(* Logix 5000 project; controller KTC_lab3 vendor 1 type 14 code 149 rev 30.11; software revision 30.00 *)

TASK MainTask (continuous, watchdog 500 ms) : MainProgram

MODULES
   Local : vendor 1 type 14 code 149 (Compact 0, rev 30.11)
      Discrete_IO : Embedded (Compact 1, rev 3.1, Output RPI 20 ms)
END_MODULES

PROGRAM MainProgram   (* main routine MainRoutine *)
VAR
   B3_1 : BOOL;   // SHUT DOWN BIT
   C5_1 : COUNTER := (ACC := 3, DN := 1);   // METAL#
   C5_2 : COUNTER := (ACC := 5, DN := 1);   // RED#
   C5_3 : COUNTER := (ACC := 3, DN := 1);   // BLACK#
   IR0 : ALIAS FOR Local:1:I.Data.0;   // done sensor
   ir07 : ALIAS FOR Local:1:O.Data.7;
   IR1 : ALIAS FOR Local:1:I.Data.3;   // NC
   IR2 : ALIAS FOR Local:1:I.Data.2;   // COLOR DETECTOR
   IR3 : ALIAS FOR Local:1:I.Data.1;   // METAL DETECTOR
   IR7 : ALIAS FOR Local:1:O.Data.7;
   PB0 : BOOL;   // PBNO reset
   PB1 : BOOL;   // PBNO run
   PB2 : BOOL;   // PBNC stop
   PB3 : BOOL;   // SHUT DOWN
   PB4 : ALIAS FOR Local:1:I.Data.11;   // RESET HW
   pb8 : ALIAS FOR Local:1:I.Data.8;   // start
   pb9 : ALIAS FOR Local:1:I.Data.9;   // stop
   PB_5 : BOOL;   // NUM RESET
   PL1 : ALIAS FOR Local:1:O.Data.9;   // stand by
   PL2 : ALIAS FOR Local:1:O.Data.8;   // LIGHT 5 run
   PL3 : ALIAS FOR Local:1:O.Data.0;   // belt
   PL4 : ALIAS FOR Local:1:O.Data.1;   // METAL ON
   PL5 : ALIAS FOR Local:1:O.Data.2;   // COLOR ON
   PL55 : ALIAS FOR Local:1:O.Data.10;   // Q1
   PL6 : ALIAS FOR Local:1:O.Data.4;   // BLACK ON
   PL66 : ALIAS FOR Local:1:O.Data.11;   // Q2
   PL7 : ALIAS FOR Local:1:O.Data.5;   // SHUT DOWN LIGHT
   sol1 : ALIAS FOR Local:1:O.Data.3;   // plunger
   SW4 : ALIAS FOR Local:1:I.Data.10;   // SWITCH 4 key switch
   T4_1 : TIMER := (PRE := 1000);
END_VAR

ROUTINE MainRoutine   (* ladder *)
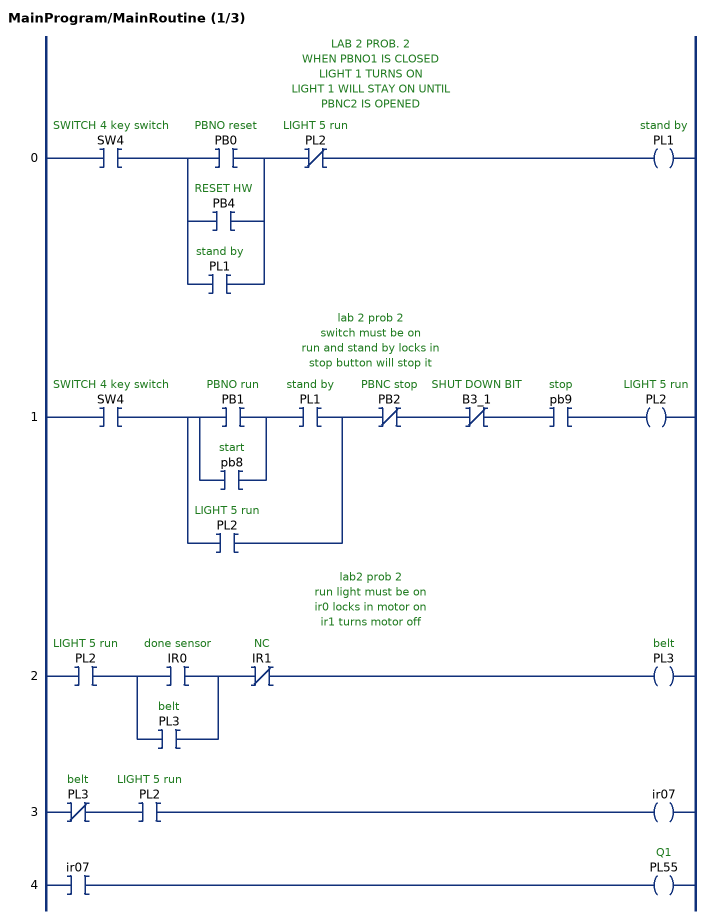
   // LAB 2 PROB. 2
   // WHEN PBNO1 IS CLOSED
   // LIGHT 1 TURNS ON
   // LIGHT 1 WILL STAY ON UNTIL
   // PBNC2 IS OPENED
   0: XIC(SW4)[[XIC(PB0) ,XIC(PB4) ] ,XIC(PL1) ]XIO(PL2)OTE(PL1);
   // lab 2 prob 2
   // switch must be on
   // run and stand by locks in
   // stop button will stop it
   1: XIC(SW4)[[XIC(PB1) ,XIC(pb8) ] XIC(PL1) ,XIC(PL2) ]XIO(PB2)XIO(B3_1)XIC(pb9)OTE(PL2);
   // lab2 prob 2
   // run light must be on
   // ir0 locks in motor on
   // ir1 turns motor off
   2: XIC(PL2)[XIC(IR0) ,XIC(PL3) ]XIO(IR1)OTE(PL3);
   3: XIO(PL3)XIC(PL2)OTE(ir07);
   4: XIC(ir07)OTE(PL55);
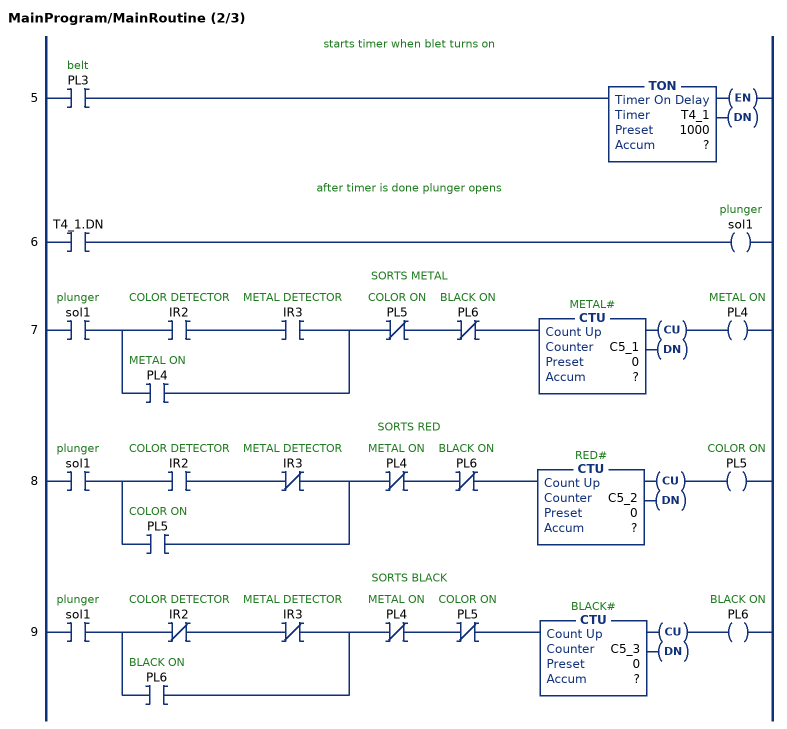
   // starts timer when blet turns on
   5: XIC(PL3)TON(T4_1,?,?);
   // after timer is done plunger opens
   6: XIC(T4_1.DN)OTE(sol1);
   // SORTS METAL
   7: XIC(sol1)[XIC(IR2) XIC(IR3) ,XIC(PL4) ]XIO(PL5)XIO(PL6)CTU(C5_1,?,?)OTE(PL4);
   // SORTS RED
   8: XIC(sol1)[XIC(IR2) XIO(IR3) ,XIC(PL5) ]XIO(PL4)XIO(PL6)CTU(C5_2,?,?)OTE(PL5);
   // SORTS BLACK
   9: XIC(sol1)[XIO(IR2) XIO(IR3) ,XIC(PL6) ]XIO(PL4)XIO(PL5)CTU(C5_3,?,?)OTE(PL6);
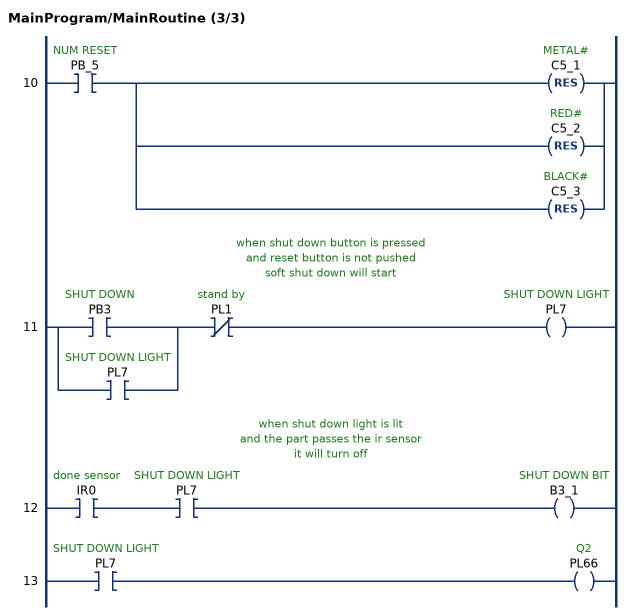
   10: XIC(PB_5)[RES(C5_1) ,RES(C5_2) ,RES(C5_3) ];
   // when shut down button is pressed
   // and reset button is not pushed
   // soft shut down will start
   11: [XIC(PB3) ,XIC(PL7) ]XIO(PL1)OTE(PL7);
   // when shut down light is lit
   // and the part passes the ir sensor
   // it will turn off
   12: XIC(IR0)XIC(PL7)OTE(B3_1);
   13: XIC(PL7)OTE(PL66);
END_ROUTINE
END_PROGRAM
